PROGRAM P002_TestAnother
VAR
	Count: INT;
	bInit: BOOL;
END_VAR

Count:=Count+2;
IF NOT bInit THEN
	bInit:=TRUE;
END_IF

END_PROGRAM

(* stored: Version 1.1.0.1, ProductVersion 3.1.4024.13
   POU P002_TestAnother: Id {c74cab12-d06d-4274-a9ed-749bfc5796e6}, SpecialFunc None *)
